Staubli VAL3: onExit.pgx

program onExit()
begin
  // save the process list
  call processList:save()
  logMsg("[KERNEL] INTERFACE:Save process list")
end
